Omron CX-Programmer project NewProject (CX-Programmer 9.03)

# PLC NewPLC1: CP1L L

## Global symbols (name address type ; comment)
0.00 BOOL  ; START
0.01 BOOL  ; STOP
0.02 BOOL  ; PHOTOSENSOR
0.03 BOOL  ; LS CCW
0.04 BOOL  ; LS CW
10.00 BOOL  ; CONVEYOR A
10.01 BOOL  ; CONVEYOR B
10.02 BOOL  ; SOLENOID CW
10.03 BOOL  ; SOLENOID CCW
1.00 BOOL  ; M
20.00 BOOL  ; GRASP

## Program NewProgram1 (cyclic task 0)

### Section Section1

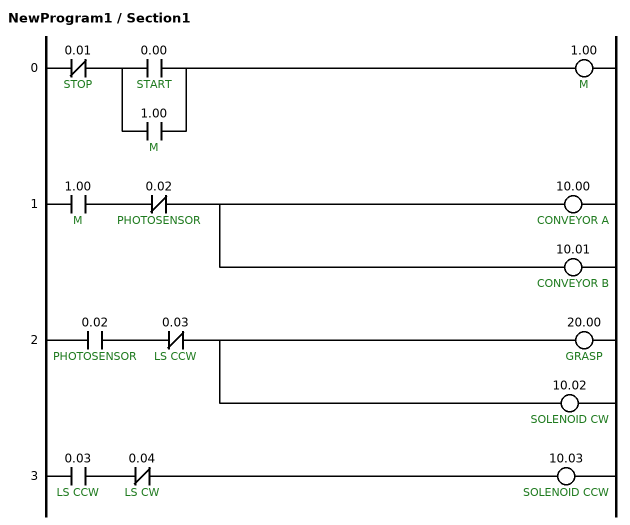
; rung 0
LDNOT 0.01  ; STOP
LD 0.00  ; START
OR 1.00  ; M
ANDLD
OUT 1.00  ; M
; rung 1
LD 1.00  ; M
ANDNOT 0.02  ; PHOTOSENSOR
OUT 10.00  ; CONVEYOR A
OUT 10.01  ; CONVEYOR B
; rung 2
LD 0.02  ; PHOTOSENSOR
ANDNOT 0.03  ; LS CCW
OUT 20.00  ; GRASP
OUT 10.02  ; SOLENOID CW
; rung 3
LD 0.03  ; LS CCW
ANDNOT 0.04  ; LS CW
OUT 10.03  ; SOLENOID CCW

### Section END
; rung 0
END(001)